SUBAPPLICATION mapping_BTN (* Subapplication Type *)
  (* Standard: 61499-2 *)
  (* Version 1.0, 2023-02-07, franz *)
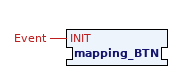
  EVENT_INPUT
    INIT;
  END_EVENT
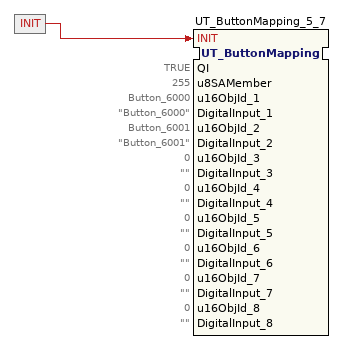
  FBS
    UT_ButtonMapping_5_7 : UT_ButtonMapping(QI := TRUE, u8SAMember := 255, u16ObjId_1 := Button_6000, DigitalInput_1 := "Button_6000", u16ObjId_2 := Button_6001, DigitalInput_2 := "Button_6001", u16ObjId_3 := 0, DigitalInput_3 := "", u16ObjId_4 := 0, DigitalInput_4 := "", u16ObjId_5 := 0, DigitalInput_5 := "", u16ObjId_6 := 0, DigitalInput_6 := "", u16ObjId_7 := 0, DigitalInput_7 := "", u16ObjId_8 := 0, DigitalInput_8 := "");
  END_FBS
  EVENT_CONNECTIONS
    INIT TO UT_ButtonMapping_5_7.INIT;
  END_CONNECTIONS
END_SUBAPPLICATION
